// TIA Portal V20 export
TYPE "LCFL_typeMTPOSLevelSiemens"
TITLE = MTP for OS level (Siemens) / MTP für OS-Level (Siemens)
// MTP data for OS level (Siemens) / MTP-Daten für OS-Level (Siemens)
   STRUCT
      mtpData : "LCFL_typeMTPOSLevel";
   END_STRUCT;
END_TYPE
